TYPE eEV_Status :
(
	NotUsed								:= -1,
	MovingForward						:= 0,
	MovingBackward						:= 1,
	MoveCompleted						:= 2,
	Timeout								:= 3,
	Error								:= 4
);
END_TYPE

(* stored: Version 1.1.0.1, ProductVersion 3.1.4024.13
   DUT eEV_Status: Id {a5731df1-87b7-434f-b8d1-f3acbcf37a04} *)
